SUBAPPLICATION Ventilsteuerung (* Subapplication Type *)
  (* Standard: 61499-2 *)
  (* Version 1.0, 2023-02-07, franz *)
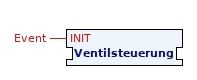
  EVENT_INPUT
    INIT;
  END_EVENT
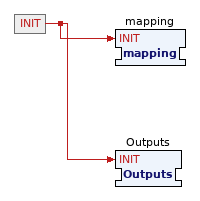
  SUBAPPS
    mapping : mapping;
    Outputs : Outputs;
  END_SUBAPPS
  EVENT_CONNECTIONS
    INIT TO mapping.INIT;
    INIT TO Outputs.INIT;
  END_CONNECTIONS
END_SUBAPPLICATION
